(* Logix 5000 project; controller SX_V040001_C001 vendor 1 type 14 code 77 rev 16.23; software revision 16.04; part 17 of 35 *)
(* tags used below, declared in another part *)
   ALL_KINDS : INT[90];
   Basic : INT;
   DRIVE : INT[32];
   G_AOutput : DINT[8];
   G_DInput : DINT[3];
   negi_param61 : DINT;
   NOTDOS : INT[6];
   PARAMETER : INT[501];
   T_CONTR_CLFA_ACLFA : TIMER;
   T_CONTR_CURR_SPEED : TIMER;
   T_CURRENT_EM_METER : TIMER;
   T_RPM_EM_METER : TIMER;
   T_TEMP_EM_METER : TIMER;
   TEMP : INT[14];
(* MainProgram, continued *)

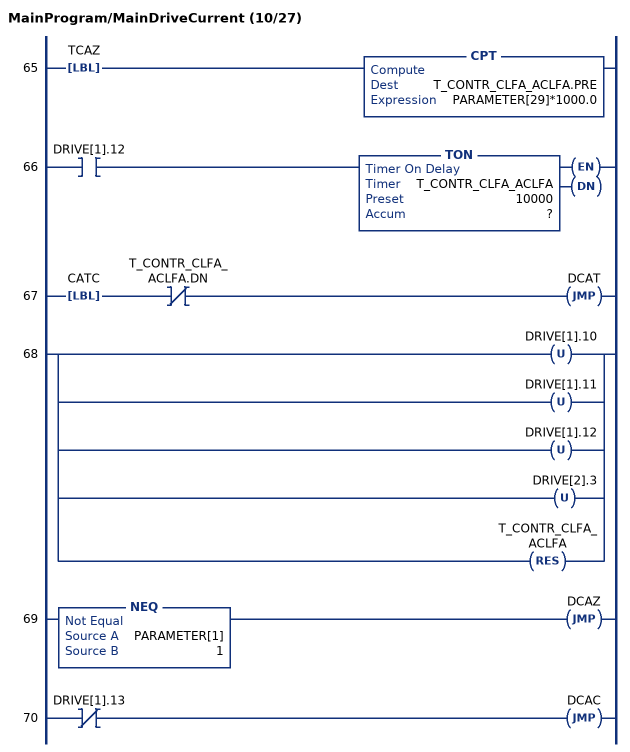
   [picture p369: MainProgram/MainDriveCurrent rungs 65-70]
   65: LBL(TCAZ)CPT(T_CONTR_CLFA_ACLFA.PRE,PARAMETER[29]*1000.0);
   66: XIC(DRIVE[1].12)TON(T_CONTR_CLFA_ACLFA,?,?);
   67: LBL(CATC)XIO(T_CONTR_CLFA_ACLFA.DN)JMP(DCAT);
   68: [OTU(DRIVE[1].10) ,OTU(DRIVE[1].11) ,OTU(DRIVE[1].12) ,OTU(DRIVE[2].3) ,RES(T_CONTR_CLFA_ACLFA) ];
   69: NEQ(PARAMETER[1],1)JMP(DCAZ);
   70: XIO(DRIVE[1].13)JMP(DCAC);
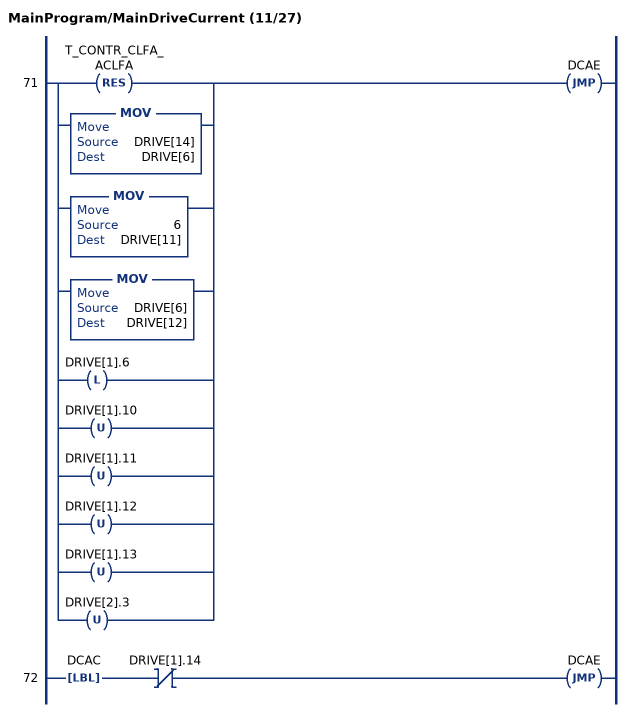
   71: [RES(T_CONTR_CLFA_ACLFA) ,MOV(DRIVE[14],DRIVE[6]) ,MOV(6,DRIVE[11]) ,MOV(DRIVE[6],DRIVE[12]) ,OTL(DRIVE[1].6) ,OTU(DRIVE[1].10) ,OTU(DRIVE[1].11) ,OTU(DRIVE[1].12) ,OTU(DRIVE[1].13) ,OTU(DRIVE[2].3) ]JMP(DCAE);
   72: LBL(DCAC)XIO(DRIVE[1].14)JMP(DCAE);
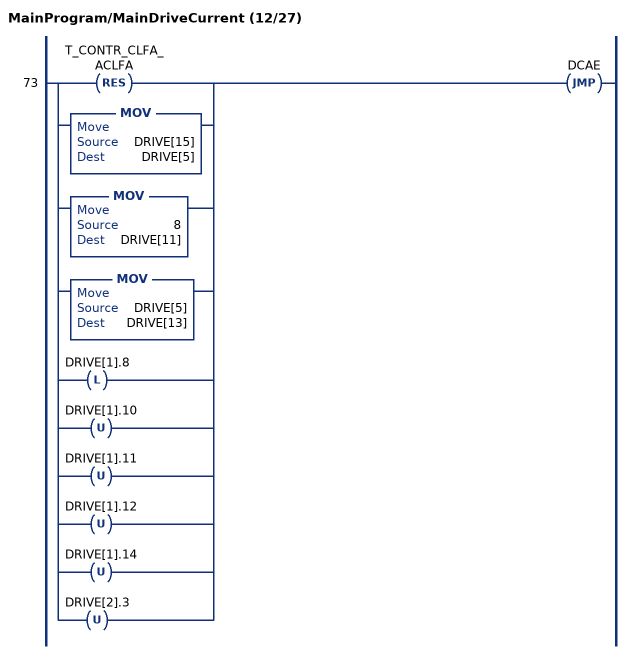
   73: [RES(T_CONTR_CLFA_ACLFA) ,MOV(DRIVE[15],DRIVE[5]) ,MOV(8,DRIVE[11]) ,MOV(DRIVE[5],DRIVE[13]) ,OTL(DRIVE[1].8) ,OTU(DRIVE[1].10) ,OTU(DRIVE[1].11) ,OTU(DRIVE[1].12) ,OTU(DRIVE[1].14) ,OTU(DRIVE[2].3) ]JMP(DCAE);
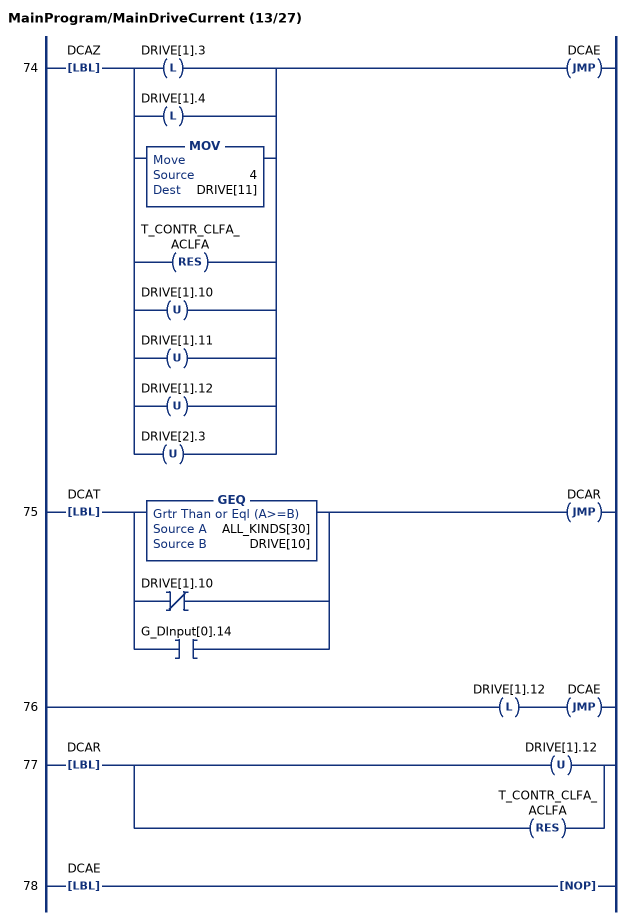
   74: LBL(DCAZ)[OTL(DRIVE[1].3) ,OTL(DRIVE[1].4) ,MOV(4,DRIVE[11]) ,RES(T_CONTR_CLFA_ACLFA) ,OTU(DRIVE[1].10) ,OTU(DRIVE[1].11) ,OTU(DRIVE[1].12) ,OTU(DRIVE[2].3) ]JMP(DCAE);
   75: LBL(DCAT)[GEQ(ALL_KINDS[30],DRIVE[10]) ,XIO(DRIVE[1].10) ,XIC(G_DInput[0].14) ]JMP(DCAR);
   76: OTL(DRIVE[1].12)JMP(DCAE);
   77: LBL(DCAR)[OTU(DRIVE[1].12) ,RES(T_CONTR_CLFA_ACLFA) ];
   78: LBL(DCAE)NOP();
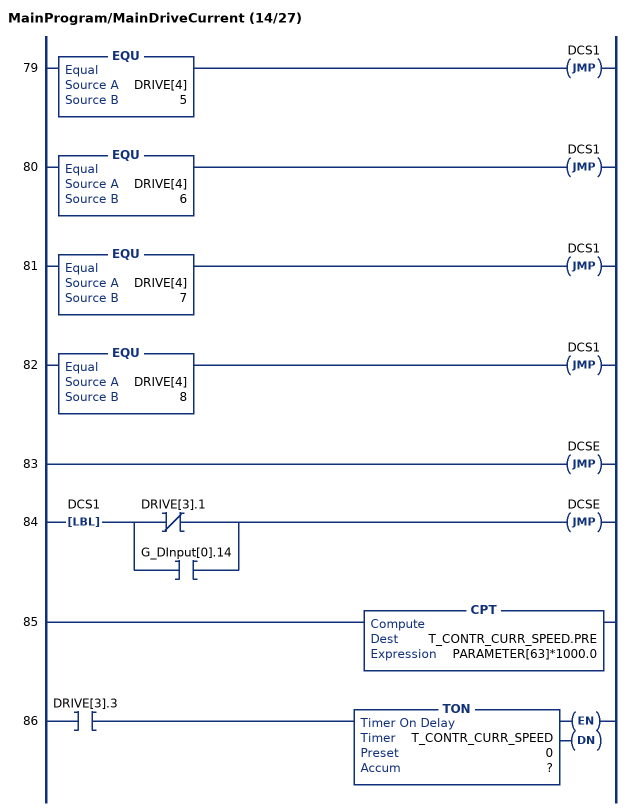
   79: EQU(DRIVE[4],5)JMP(DCS1);
   80: EQU(DRIVE[4],6)JMP(DCS1);
   81: EQU(DRIVE[4],7)JMP(DCS1);
   82: EQU(DRIVE[4],8)JMP(DCS1);
   83: JMP(DCSE);
   84: LBL(DCS1)[XIO(DRIVE[3].1) ,XIC(G_DInput[0].14) ]JMP(DCSE);
   85: CPT(T_CONTR_CURR_SPEED.PRE,PARAMETER[63]*1000.0);
   86: XIC(DRIVE[3].3)TON(T_CONTR_CURR_SPEED,?,?);
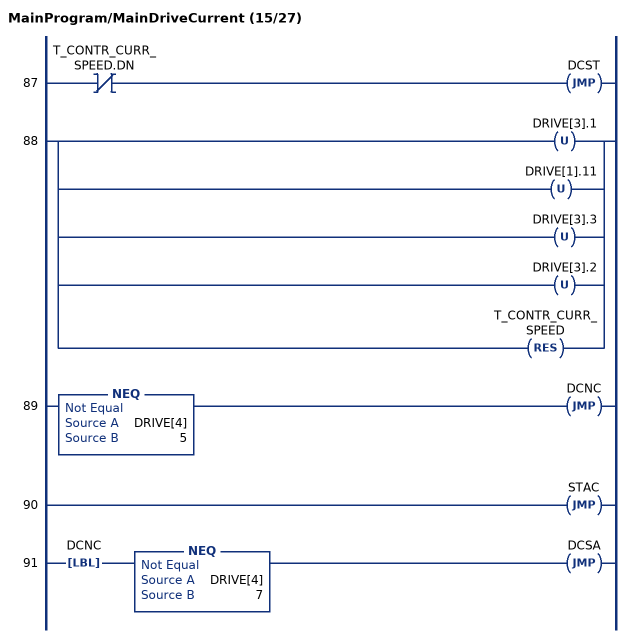
   87: XIO(T_CONTR_CURR_SPEED.DN)JMP(DCST);
   88: [OTU(DRIVE[3].1) ,OTU(DRIVE[1].11) ,OTU(DRIVE[3].3) ,OTU(DRIVE[3].2) ,RES(T_CONTR_CURR_SPEED) ];
   89: NEQ(DRIVE[4],5)JMP(DCNC);
   90: JMP(STAC);
   91: LBL(DCNC)NEQ(DRIVE[4],7)JMP(DCSA);
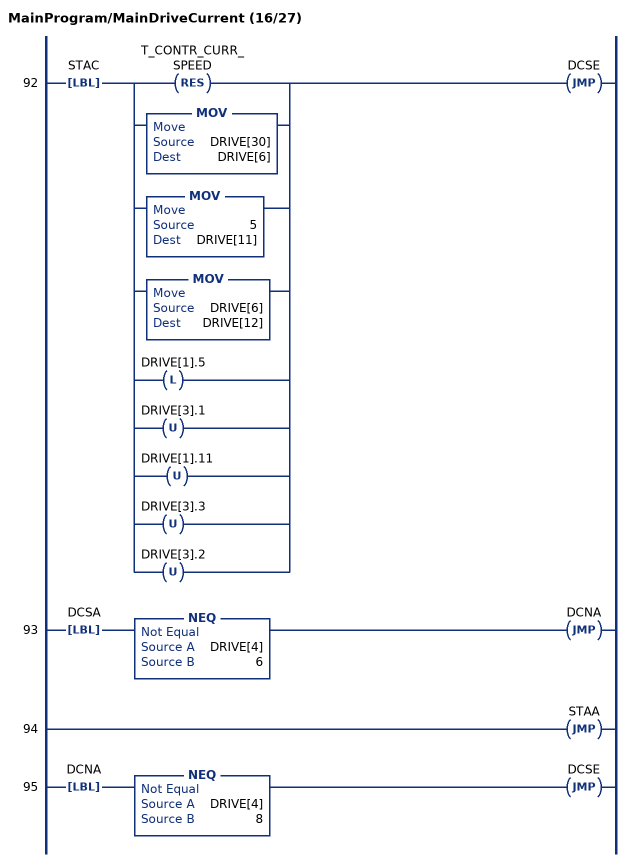
   92: LBL(STAC)[RES(T_CONTR_CURR_SPEED) ,MOV(DRIVE[30],DRIVE[6]) ,MOV(5,DRIVE[11]) ,MOV(DRIVE[6],DRIVE[12]) ,OTL(DRIVE[1].5) ,OTU(DRIVE[3].1) ,OTU(DRIVE[1].11) ,OTU(DRIVE[3].3) ,OTU(DRIVE[3].2) ]JMP(DCSE);
   93: LBL(DCSA)NEQ(DRIVE[4],6)JMP(DCNA);
   94: JMP(STAA);
   95: LBL(DCNA)NEQ(DRIVE[4],8)JMP(DCSE);
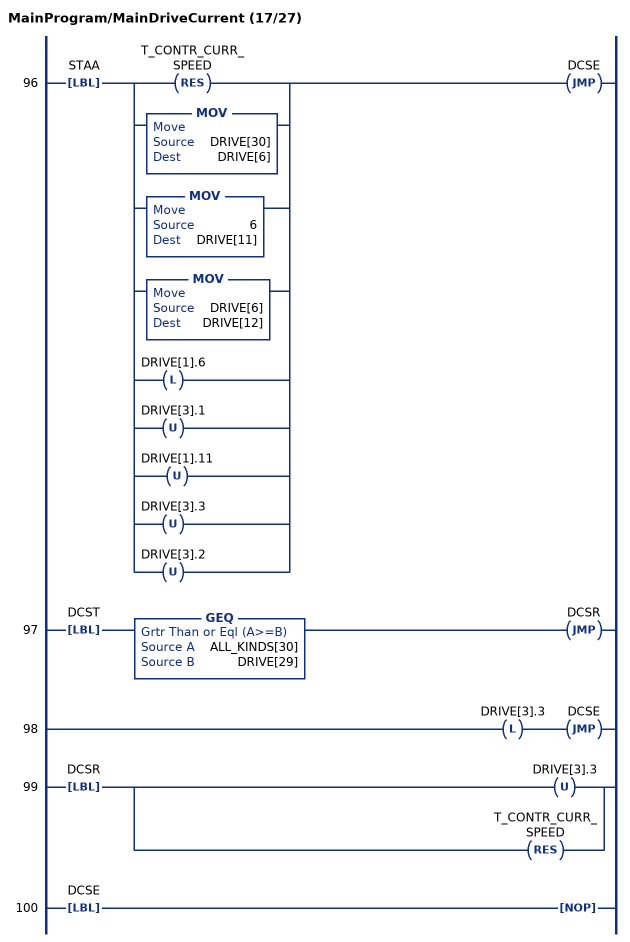
   96: LBL(STAA)[RES(T_CONTR_CURR_SPEED) ,MOV(DRIVE[30],DRIVE[6]) ,MOV(6,DRIVE[11]) ,MOV(DRIVE[6],DRIVE[12]) ,OTL(DRIVE[1].6) ,OTU(DRIVE[3].1) ,OTU(DRIVE[1].11) ,OTU(DRIVE[3].3) ,OTU(DRIVE[3].2) ]JMP(DCSE);
   97: LBL(DCST)GEQ(ALL_KINDS[30],DRIVE[29])JMP(DCSR);
   98: OTL(DRIVE[3].3)JMP(DCSE);
   99: LBL(DCSR)[OTU(DRIVE[3].3) ,RES(T_CONTR_CURR_SPEED) ];
   100: LBL(DCSE)NOP();
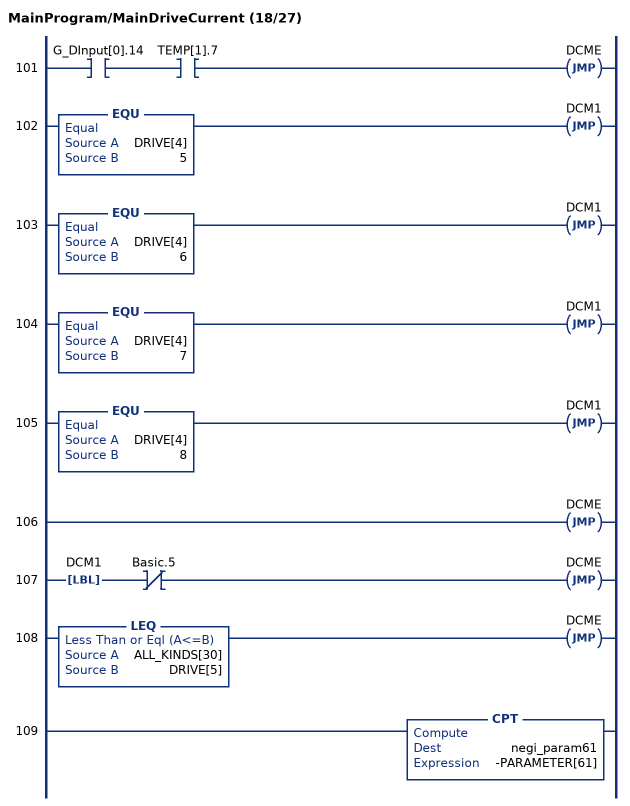
   101: XIC(G_DInput[0].14)XIC(TEMP[1].7)JMP(DCME);
   102: EQU(DRIVE[4],5)JMP(DCM1);
   103: EQU(DRIVE[4],6)JMP(DCM1);
   104: EQU(DRIVE[4],7)JMP(DCM1);
   105: EQU(DRIVE[4],8)JMP(DCM1);
   106: JMP(DCME);
   107: LBL(DCM1)XIO(Basic.5)JMP(DCME);
   108: LEQ(ALL_KINDS[30],DRIVE[5])JMP(DCME);
   109: CPT(negi_param61,-PARAMETER[61]);
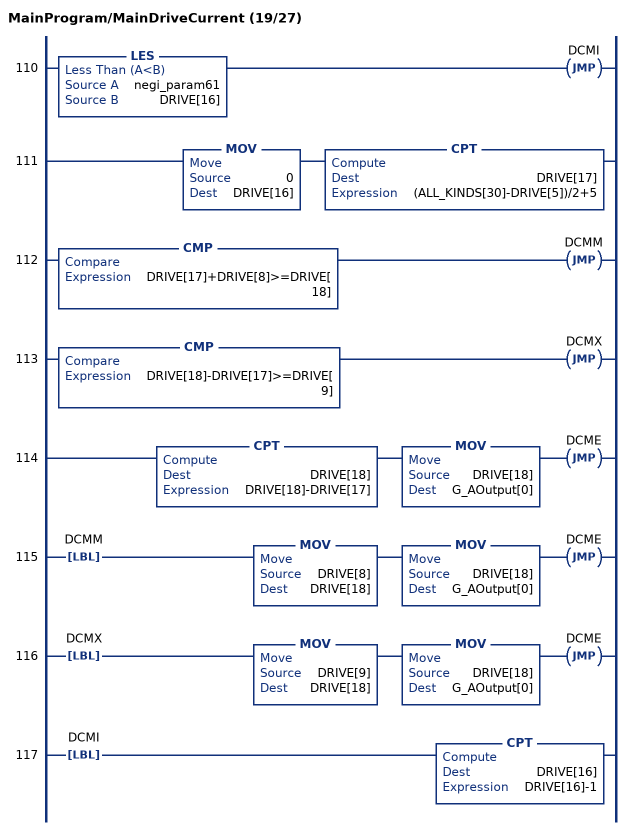
   110: LES(negi_param61,DRIVE[16])JMP(DCMI);
   111: MOV(0,DRIVE[16])CPT(DRIVE[17],(ALL_KINDS[30]-DRIVE[5])/2+5);
   112: CMP(DRIVE[17]+DRIVE[8]>=DRIVE[18])JMP(DCMM);
   113: CMP(DRIVE[18]-DRIVE[17]>=DRIVE[9])JMP(DCMX);
   114: CPT(DRIVE[18],DRIVE[18]-DRIVE[17])MOV(DRIVE[18],G_AOutput[0])JMP(DCME);
   115: LBL(DCMM)MOV(DRIVE[8],DRIVE[18])MOV(DRIVE[18],G_AOutput[0])JMP(DCME);
   116: LBL(DCMX)MOV(DRIVE[9],DRIVE[18])MOV(DRIVE[18],G_AOutput[0])JMP(DCME);
   117: LBL(DCMI)CPT(DRIVE[16],DRIVE[16]-1);
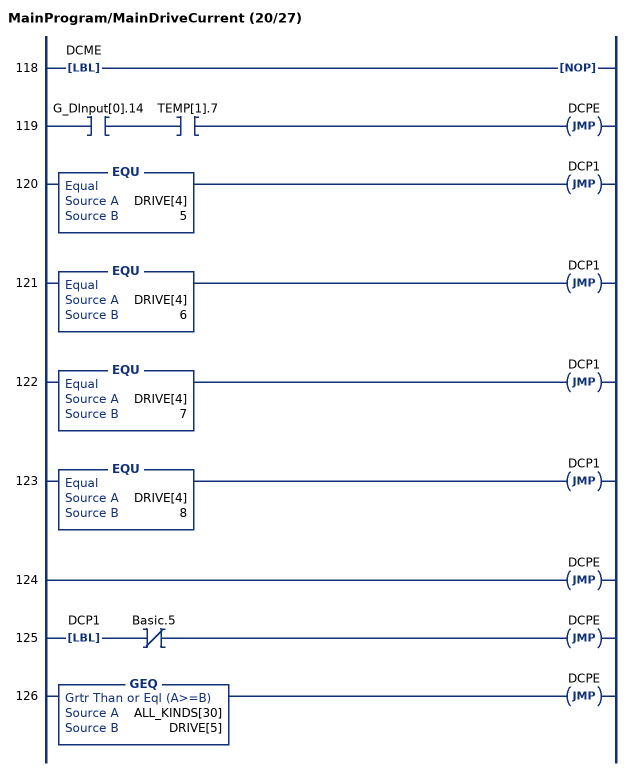
   118: LBL(DCME)NOP();
   119: XIC(G_DInput[0].14)XIC(TEMP[1].7)JMP(DCPE);
   120: EQU(DRIVE[4],5)JMP(DCP1);
   121: EQU(DRIVE[4],6)JMP(DCP1);
   122: EQU(DRIVE[4],7)JMP(DCP1);
   123: EQU(DRIVE[4],8)JMP(DCP1);
   124: JMP(DCPE);
   125: LBL(DCP1)XIO(Basic.5)JMP(DCPE);
   126: GEQ(ALL_KINDS[30],DRIVE[5])JMP(DCPE);
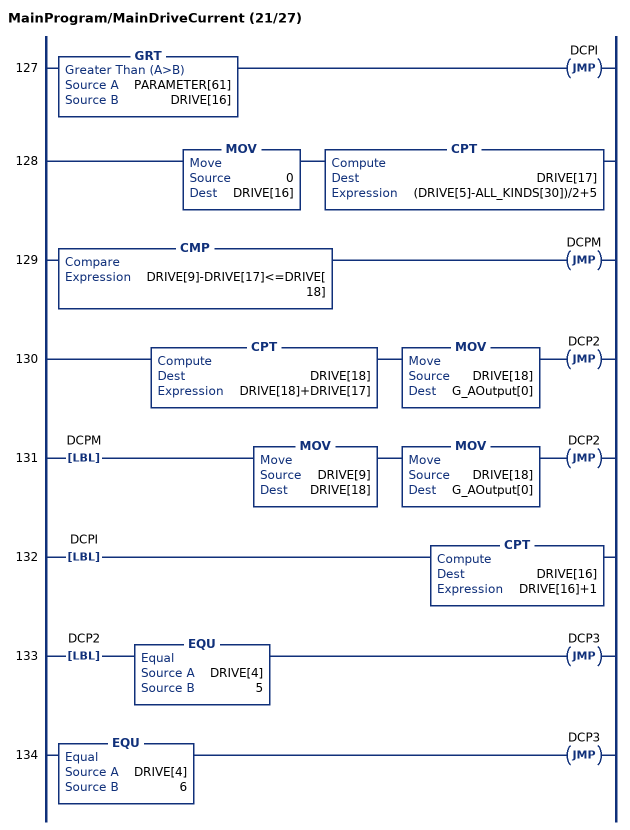
   127: GRT(PARAMETER[61],DRIVE[16])JMP(DCPI);
   128: MOV(0,DRIVE[16])CPT(DRIVE[17],(DRIVE[5]-ALL_KINDS[30])/2+5);
   129: CMP(DRIVE[9]-DRIVE[17]<=DRIVE[18])JMP(DCPM);
   130: CPT(DRIVE[18],DRIVE[18]+DRIVE[17])MOV(DRIVE[18],G_AOutput[0])JMP(DCP2);
   131: LBL(DCPM)MOV(DRIVE[9],DRIVE[18])MOV(DRIVE[18],G_AOutput[0])JMP(DCP2);
   132: LBL(DCPI)CPT(DRIVE[16],DRIVE[16]+1);
   133: LBL(DCP2)EQU(DRIVE[4],5)JMP(DCP3);
   134: EQU(DRIVE[4],6)JMP(DCP3);
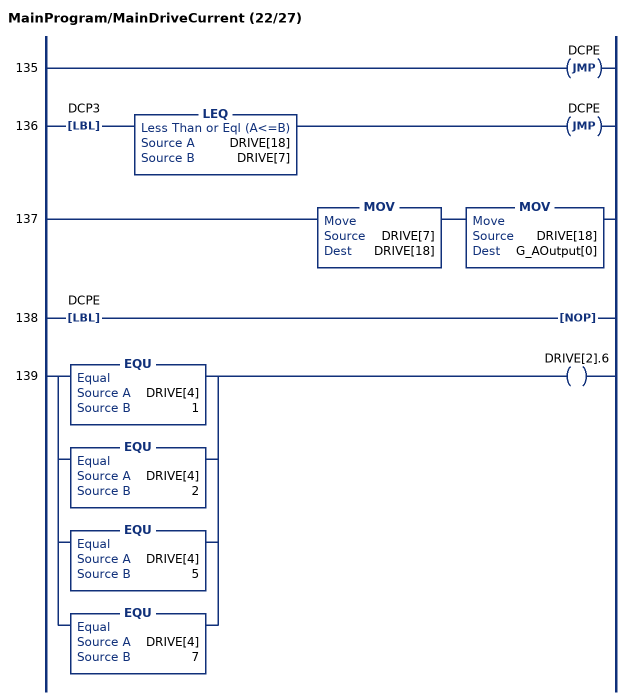
   135: JMP(DCPE);
   136: LBL(DCP3)LEQ(DRIVE[18],DRIVE[7])JMP(DCPE);
   137: MOV(DRIVE[7],DRIVE[18])MOV(DRIVE[18],G_AOutput[0]);
   138: LBL(DCPE)NOP();
   139: [EQU(DRIVE[4],1) ,EQU(DRIVE[4],2) ,EQU(DRIVE[4],5) ,EQU(DRIVE[4],7) ]OTE(DRIVE[2].6);
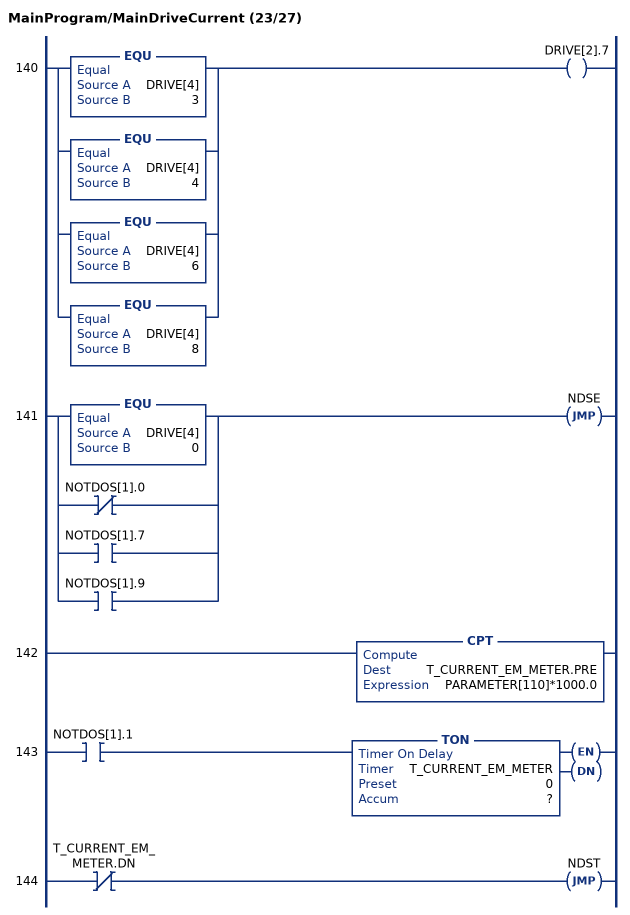
   140: [EQU(DRIVE[4],3) ,EQU(DRIVE[4],4) ,EQU(DRIVE[4],6) ,EQU(DRIVE[4],8) ]OTE(DRIVE[2].7);
   141: [EQU(DRIVE[4],0) ,XIO(NOTDOS[1].0) ,XIC(NOTDOS[1].7) ,XIC(NOTDOS[1].9) ]JMP(NDSE);
   142: CPT(T_CURRENT_EM_METER.PRE,PARAMETER[110]*1000.0);
   143: XIC(NOTDOS[1].1)TON(T_CURRENT_EM_METER,?,?);
   144: XIO(T_CURRENT_EM_METER.DN)JMP(NDST);
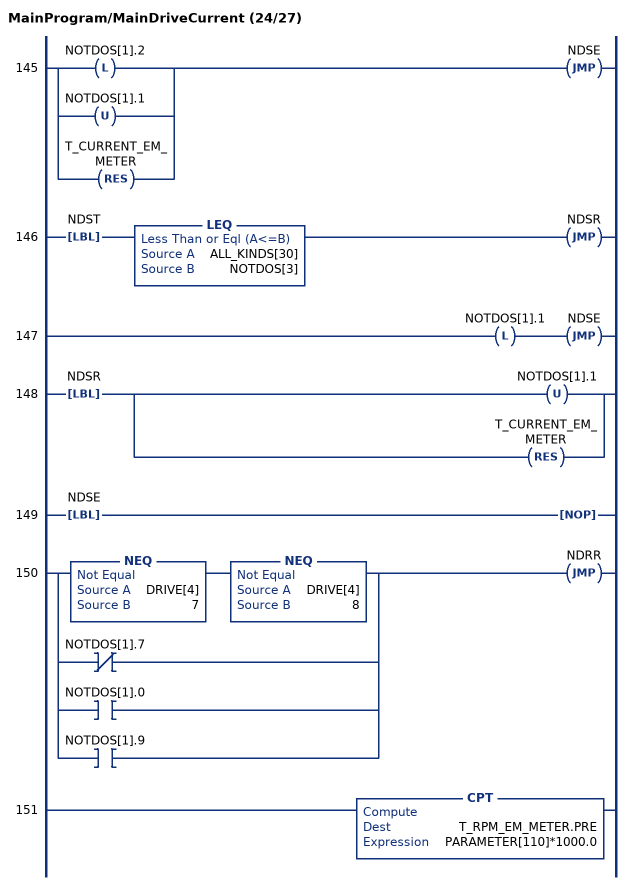
   145: [OTL(NOTDOS[1].2) ,OTU(NOTDOS[1].1) ,RES(T_CURRENT_EM_METER) ]JMP(NDSE);
   146: LBL(NDST)LEQ(ALL_KINDS[30],NOTDOS[3])JMP(NDSR);
   147: OTL(NOTDOS[1].1)JMP(NDSE);
   148: LBL(NDSR)[OTU(NOTDOS[1].1) ,RES(T_CURRENT_EM_METER) ];
   149: LBL(NDSE)NOP();
   150: [NEQ(DRIVE[4],7) NEQ(DRIVE[4],8) ,XIO(NOTDOS[1].7) ,XIC(NOTDOS[1].0) ,XIC(NOTDOS[1].9) ]JMP(NDRR);
   151: CPT(T_RPM_EM_METER.PRE,PARAMETER[110]*1000.0);
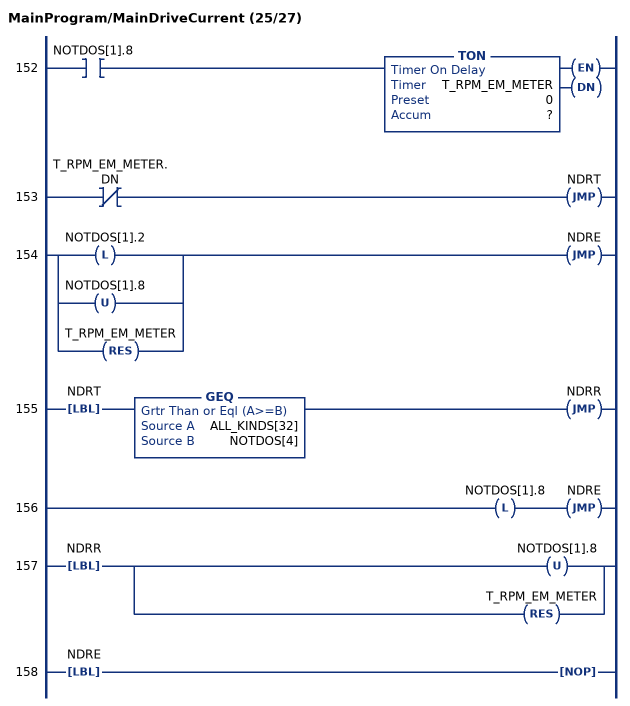
   152: XIC(NOTDOS[1].8)TON(T_RPM_EM_METER,?,?);
   153: XIO(T_RPM_EM_METER.DN)JMP(NDRT);
   154: [OTL(NOTDOS[1].2) ,OTU(NOTDOS[1].8) ,RES(T_RPM_EM_METER) ]JMP(NDRE);
   155: LBL(NDRT)GEQ(ALL_KINDS[32],NOTDOS[4])JMP(NDRR);
   156: OTL(NOTDOS[1].8)JMP(NDRE);
   157: LBL(NDRR)[OTU(NOTDOS[1].8) ,RES(T_RPM_EM_METER) ];
   158: LBL(NDRE)NOP();
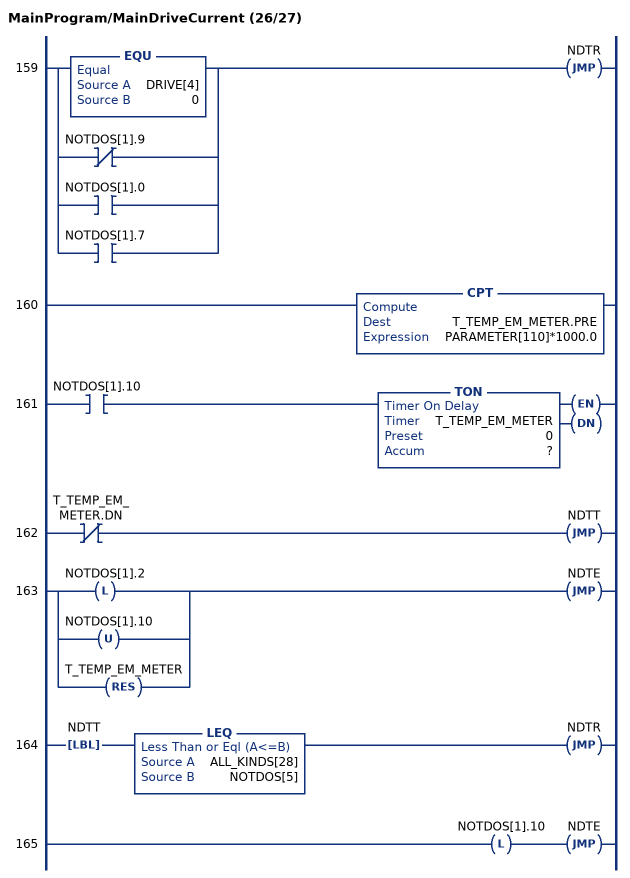
   159: [EQU(DRIVE[4],0) ,XIO(NOTDOS[1].9) ,XIC(NOTDOS[1].0) ,XIC(NOTDOS[1].7) ]JMP(NDTR);
   160: CPT(T_TEMP_EM_METER.PRE,PARAMETER[110]*1000.0);
   161: XIC(NOTDOS[1].10)TON(T_TEMP_EM_METER,?,?);
   162: XIO(T_TEMP_EM_METER.DN)JMP(NDTT);
   163: [OTL(NOTDOS[1].2) ,OTU(NOTDOS[1].10) ,RES(T_TEMP_EM_METER) ]JMP(NDTE);
   164: LBL(NDTT)LEQ(ALL_KINDS[28],NOTDOS[5])JMP(NDTR);
   165: OTL(NOTDOS[1].10)JMP(NDTE);
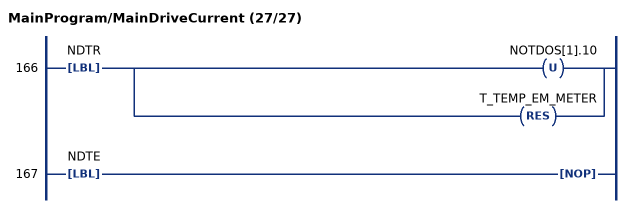
   166: LBL(NDTR)[OTU(NOTDOS[1].10) ,RES(T_TEMP_EM_METER) ];
   167: LBL(NDTE)NOP();
END_ROUTINE
